TYPE ST_NestedTypes03 :
STRUCT
	stPytmcTypes : ST_PytmcTypes;
	stNestedTypes : ST_NestedTypes04;
END_STRUCT
END_TYPE

(* stored: Version 1.1.0.1, ProductVersion 3.1.4026.12
   DUT ST_NestedTypes03: Id {345e57fa-e807-478e-b3cf-d8b15fd4a7e4} *)
